// TIA Portal V17 export
// export: Created 2025-03-13T10:31:24.9988544Z, ExportSetting WithDefaults, DisplayName Totally Integrated Automation Portal, DisplayVersion V17 Update 8, DisplayName TIA Portal Openness, DisplayVersion V17 Update 8, DisplayName TIA Portal Version Control Interface, DisplayVersion V17, DisplayName SINAMICS Startdrive Advanced, DisplayVersion V17 SP2, DisplayName SINAMICS Startdrive G110M, G120, G120C, G120D, G120P, G115D, DisplayVersion V17 SP2, DisplayName SINAMICS Startdrive G130, G150, S120, S150, SINAMICS MV, S210, DisplayVersion V17 SP2, DisplayName STEP 7 Professional, DisplayVersion V17 Update 8, DisplayName SINUMERIK ONE STEP 7 Toolbox, DisplayVersion V17 Update 12, DisplayName SINUMERIK 840D sl STEP 7 Toolbox, DisplayVersion V17 Update 12, DisplayName STEP 7 Safety, DisplayVersion V17 Update 6, DisplayName WinCC Advanced, DisplayVersion V17 Update 8
TYPE "CRASH_BORE_MEAS"
// stored: IsFailsafeCompliant false
   STRUCT
      MEAS_1 : Real;   // MEASUREMENT POINT 1
      MEAS_2 : Real;   // MEASUREMENT POINT 2
      MEAS_3 : Real;   // MEASUREMENT POINT 3
      MEAS_4 : Real;   // MEASUREMENT POINT 4
      MEAS_5 : Real;   // MEASUREMENT POINT 5
      MEAS_6 : Real;   // MEASUREMENT POINT 6
      MEAS_7X : Real;   // MEASUREMENT POINT 7X
      MEAS_7Y : Real;   // MEASUREMENT POINT 7Y
      MEAS_8X : Real;   // MEASUREMENT POINT 8X
      MEAS_8Y : Real;   // MEASUREMENT POINT 8Y
   END_STRUCT;
END_TYPE
